// TIA Portal V17 export
// export: Created 2025-03-10T13:12:14.7117036Z, ExportSetting WithDefaults, DisplayName Totally Integrated Automation Portal, DisplayVersion V17 Update 8, DisplayName TIA Portal Openness, DisplayVersion V17 Update 8, DisplayName TIA Portal Version Control Interface, DisplayVersion V17, DisplayName SINAMICS Startdrive Advanced, DisplayVersion V17 SP2, DisplayName SINAMICS Startdrive G110M, G120, G120C, G120D, G120P, G115D, DisplayVersion V17 SP2, DisplayName SINAMICS Startdrive G130, G150, S120, S150, SINAMICS MV, S210, DisplayVersion V17 SP2, DisplayName STEP 7 Professional, DisplayVersion V17 Update 8, DisplayName SINUMERIK ONE STEP 7 Toolbox, DisplayVersion V17 Update 12, DisplayName SINUMERIK 840D sl STEP 7 Toolbox, DisplayVersion V17 Update 12, DisplayName STEP 7 Safety, DisplayVersion V17 Update 6, DisplayName WinCC Advanced, DisplayVersion V17 Update 8
TYPE "MR_J4_TN_Input"
// stored: IsFailsafeCompliant false
   STRUCT
      Input : Struct
         "I_mode operation_B1" : Byte;
         "I_mode operation_B2" : Byte;
         I_SW_B8 : Bool;
         I_SW_B9_RM : Bool;
         I_SW_B10_TR : Bool;
         I_SW_B11_ILA : Bool;
         I_SW_B12_SPoint : Bool;
         I_SW_B13_FError : Bool;
         I_SW_B14 : Bool;
         I_SW_B15 : Bool;
         I_SW_B0_RTSO : Bool;
         I_SW_B1_SO : Bool;
         I_SW_B2_0E : Bool;
         I_SW_B3_Fault : Bool;
         I_SW_B4_VE : Bool;
         I_SW_B5_QS : Bool;
         I_SW_B6_SOD : Bool;
         I_SW_B7_Warning : Bool;
         I_SDO1_B8 : Bool;
         I_SDO1_B9 : Bool;
         I_SDO1_B10 : Bool;
         I_SDO1_B11 : Bool;
         I_SDO1_B12_S_INP : Bool;
         I_SDO1_B13_S_TLC : Bool;
         I_SDO1_B14_S_ABSV : Bool;
         I_SDO1_B15_S_BWNG : Bool;
         I_SDO1_B0 : Bool;
         I_SDO1_B1 : Bool;
         I_SDO1_B2_S_SA : Bool;
         I_SDO1_B3_S_MBR : Bool;
         I_SDO1_B4_S_CDPS : Bool;
         I_SDO1_B5_S_CLD : Bool;
         I_SDO1_B6 : Bool;
         I_SDO1_B7 : Bool;
         I_SDO2_B8_S_PC : Bool;
         I_SDO2_B9 : Bool;
         I_SDO2_B10_S_DB : Bool;
         I_SDO2_B11 : Bool;
         I_SDO2_B12 : Bool;
         I_SDO2_B13 : Bool;
         I_SDO2_B14 : Bool;
         I_SDO2_B15_S_ZP2 : Bool;
         I_SDO2_B0_S_ZPAS : Bool;
         I_SDO2_B1 : Bool;
         I_SDO2_B2 : Bool;
         I_SDO2_B3_S_ZSP : Bool;
         I_SDO2_B4_S_VLC : Bool;
         I_SDO2_B5 : Bool;
         I_SDO2_B6_S_IPF : Bool;
         I_SDO2_B7 : Bool;
         I_SDO3 : Word;
         "I_Torque actual" : Int;
         "I_Digital input" : DWord;
         "I_Posicion actual" : DInt;
         "I_Velocity actual" : DInt;
         "I_Following error" : DInt;
         "I_Touch probe_pos1 pos" : DInt;
         "I_Touch_probe_pos1 neg" : DInt;
         "I_Touch_probe_pos2 pos" : DInt;
         "I_Touch_probe_pos2 neg" { ExternalAccessible := 'False'; ExternalVisible := 'False'; ExternalWritable := 'False'} : DInt;
         I_Touch_probe_status : Int;
         I_reserved : Word;
      END_STRUCT;
   END_STRUCT;
END_TYPE
